Fanuc KAREL source: ka00105.KL

PROGRAM KA00105
%NOLOCKGROUP
VAR
SRC : VECTOR;DST : VECTOR
BEGIN
--
SRC.X=1.0
DST=SRC
END KA00105
